// TIA Portal V18 export
TYPE "Station"
   STRUCT
      SensorA : Bool;
      SensorB : Bool;
      SensorC : Bool;
      SensorD : Bool;
      IsEmpty : Bool;
      IsOccupied : Bool;
      Number : Bool;
   END_STRUCT;
END_TYPE
